ABB RobotStudio station: 实验二加基本自定义动作.rspag

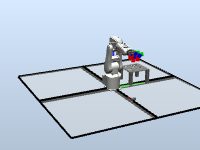
--- station ---
Station PartC (saved by RobotStudio 6.8.8148.134)
Controller System2
  mechanical unit ROB_1: IRB120_3_58__01, 6 joints, base frame (0, 0, 0) mm
Layout (positions relative to the parent item):
  - IRB120_3_58__01 [mechanism, from Robots\IRB120_3_58_G_01.rslib] at (0, 0, 0) mm; joint values [0.0061, 0.1198, 0.0289, 0.0001, -0.1484, -0.0004] (rad or m)
  - SmartComponent_1 [smart component] at (413.29, 2.5, 582.55) mm, rotated rx -130.44 ry 89.98 rz -130.09 deg
      signals: DI GET, DO FINISH, DI GET1, DO FINISH1
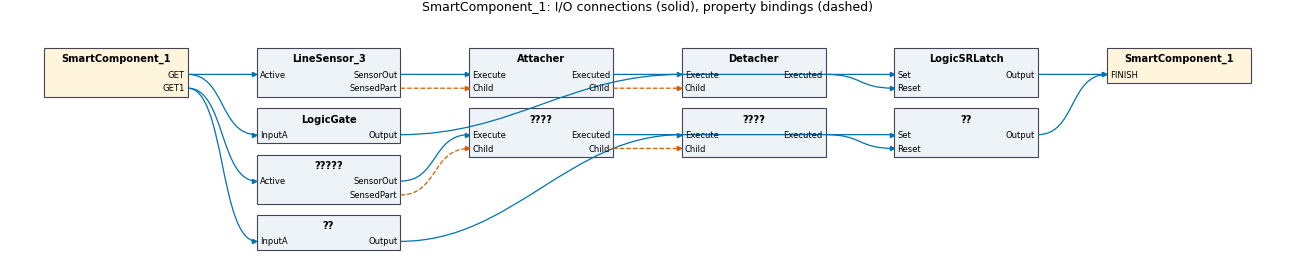
      connections:
        SmartComponent_1.GET -> LineSensor_3.Active
        SmartComponent_1.GET -> LogicGate.InputA
        LineSensor_3.SensorOut -> Attacher.Execute
        LogicGate.Output -> Detacher.Execute
        Attacher.Executed -> LogicSRLatch.Set
        Detacher.Executed -> LogicSRLatch.Reset
        LogicSRLatch.Output -> SmartComponent_1.FINISH
        SmartComponent_1.GET1 -> 吸盘传感器.Active
        SmartComponent_1.GET1 -> 吸盘.InputA
        吸盘传感器.SensorOut -> 吸盘安装.Execute
        吸盘.Output -> 吸盘拆除.Execute
        吸盘安装.Executed -> 吸盘.Set
        吸盘拆除.Executed -> 吸盘.Reset
        吸盘.Output -> SmartComponent_1.FINISH
        LineSensor_3.SensedPart => Attacher.Child
        Attacher.Child => Detacher.Child
        吸盘传感器.SensedPart => 吸盘安装.Child
        吸盘安装.Child => 吸盘拆除.Child
    - LineSensor_3 [smart component, from Components\LineSensor.rslib] at (-22.5, 0, 83.55) mm
        properties: Start=[0.0150000000000009 -0.000761999999999613 0.00306099999999904]; End=[-0.0249959999999991 0.00111800000000039 0.00431999999999905]; Radius=0.005; SensedPart=TCP-练习笔; SensedPoint=[-0.0910473251342774 0.454946044921875 0.202438980102539]
      - _sensorPart_ [part]
    - Attacher [smart component, from Components\Attacher.rslib]
        properties: Parent=SmartComponent_1; Flange=0; Child=TCP-练习笔; Mount=false; Offset=[0 0 0]; Orientation=[0 0 0]
    - Detacher [smart component, from Components\Detacher.rslib]
        properties: Child=TCP-练习笔; KeepPosition=true
    - LogicGate [smart component, from Components\LogicGate.rslib]
        properties: Operator=NOT; Delay=0
    - LogicSRLatch [smart component, from Components\LogicSRLatch.rslib]
    - My_Mechanism [mechanism] at (0, 0, 0) mm; joint values [0.01] (rad or m)
        TCP tool1 at (15.5, 0, 69.3) mm
        TCP tool2 at (-22.5, 0, 83.55) mm
        TCP tool3 at (-22.5, 0, 160.55) mm
        links: L1, L2
    - 吸盘传感器 [smart component, from Components\LineSensor.rslib] at (15.5, 0, 69.3) mm
        properties: Start=[-9.24038488097009E-05 3.65283253372798E-07 6.91615849535143E-07]; End=[0.00653224996369399 -0.000166814998235508 -0.000226620747395823]; Radius=0.005; SensedPart=部件_2; SensedPoint=[0.465495025634766 0.029700740814209 0.03]
      - _sensorPart_ [part]
    - 吸盘安装 [smart component, from Components\Attacher.rslib]
        properties: Parent=SmartComponent_1; Flange=0; Child=部件_2; Mount=false; Offset=[0 0 0]; Orientation=[0 0 0]
    - 吸盘拆除 [smart component, from Components\Detacher.rslib]
        properties: Child=部件_2; KeepPosition=true
    - 吸盘 [smart component, from Components\LogicGate.rslib]
        properties: Operator=NOT; Delay=0
    - 吸盘 [smart component, from Components\LogicSRLatch.rslib]
  - 部件_2 [part] at (0, 0, 0) mm
  - TCP_Table [part]
  - TCP-练习笔 [part] at (0, 0, 0) mm
  - 框架_1 [frame] at (15.5, 0, 69.3) mm
  - 框架_2 [frame] at (-22.5, 0, 83.55) mm
  - 框架_3 [frame] at (-22.5, 0, 160.55) mm
Attachment: My_Mechanism is attached to IRB120_3_58__01 / Link6
Attachment: SmartComponent_1 is attached to IRB120_3_58__01 / Link6
Attachment: LineSensor_3 is attached to My_Mechanism / L1
Attachment: 吸盘传感器 is attached to My_Mechanism / L1
EventTableEntry 2443: Group=, Trigger=DO_007 2444, Actions=[EventTableActionMechanicalPose 2445], Comment=, ActivationMode=2, Cyclic=false
EventTableTriggerIO 2444: IOValue=[1], IRC5Controller=? -1, Operator=0, SignalSource=System2 2451
EventTableActionMechanicalPose 2445: VirtualSignal=, Mechanism=My_Mechanism 980, ToPoseName=SyncPosition, VirtualSignalValue=[1]
EventTableEntry 2446: Group=, Trigger=DO_007 2447, Actions=[EventTableActionMechanicalPose 2448], Comment=, ActivationMode=2, Cyclic=false
EventTableTriggerIO 2447: IOValue=[0], IRC5Controller=? -1, Operator=0, SignalSource=System2 2451
EventTableActionMechanicalPose 2448: VirtualSignal=, Mechanism=My_Mechanism 980, ToPoseName=HomePosition, VirtualSignalValue=[1]
Station logic (signal -> signal, property => property):
  System2.DO_007 -> SmartComponent_1.GET
  System2.DO_0077 -> SmartComponent_1.GET1
Targets, tools, work objects and paths stored in the station and not in the controller backup, written as RAPID:
! task T_ROB1
MODULE CalibData
  PERS tooldata tool1:=[TRUE,[[15.5,0,69.3],[1,0,0,0]],[1,[0,0,1],[1,0,0,0],0,0,0]];
  PERS tooldata tool2:=[TRUE,[[-22.5,0,83.554],[1,0,0,0]],[1,[0,0,1],[1,0,0,0],0,0,0]];
  PERS tooldata tool3:=[TRUE,[[-22.5,0,160.554],[1,0,0,0]],[1,[0,0,1],[1,0,0,0],0,0,0]];
  PERS tooldata Tooldata_4:=[TRUE,[[15.5,0,69.3],[1,0,0,0]],[1,[0,0,1],[1,0,0,0],0,0,0]];
  PERS tooldata Tooldata_5:=[TRUE,[[-22.5,0,83.554],[1,0,0,0]],[1,[0,0,1],[1,0,0,0],0,0,0]];
  PERS tooldata Tooldata_6:=[TRUE,[[-22.5,0,160.554],[1,0,0,0]],[1,[0,0,1],[1,0,0,0],0,0,0]];
ENDMODULE


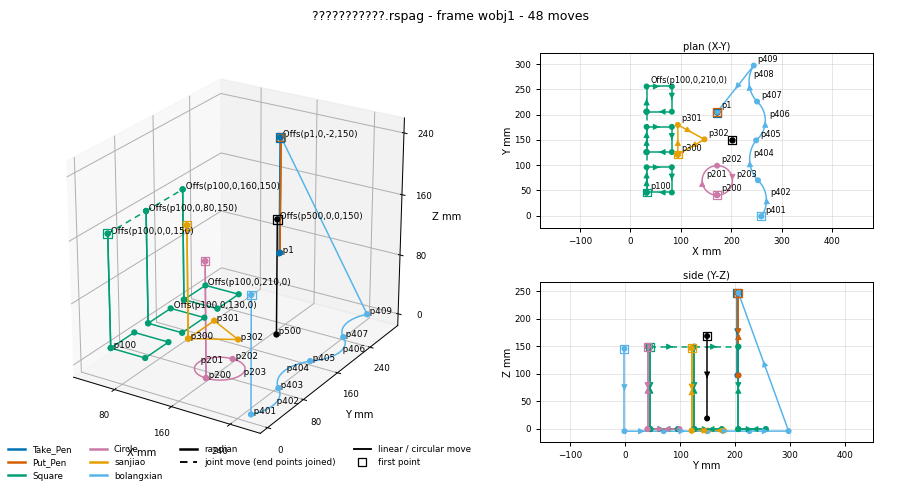
[picture p0: tool path of 实验二加基本自定义动作.rspag in frame wobj1, 48 of 55 moves have a stored position in this frame; points joined in program order, loops and branches not executed]
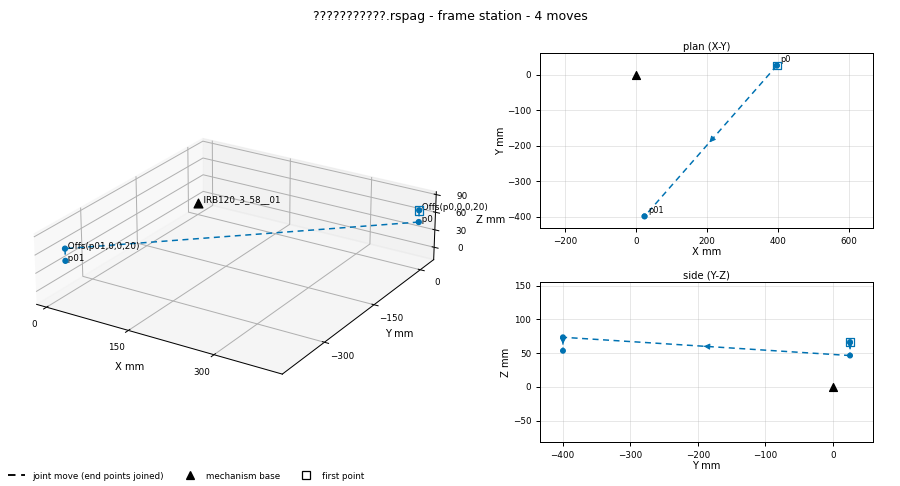
[picture p1: tool path of 实验二加基本自定义动作.rspag in frame station, 4 of 55 moves have a stored position in this frame; points joined in program order, loops and branches not executed]
--- Backups/System2/RAPID/TASK1/PROGMOD/Module1.mod ---
MODULE Module1
	TASK PERS loaddata load1:=[1,[0,0,50],[1,0,0,0],0,0,0];
	CONST robtarget p1:=[[172.01,205.77,97.31],[0.00112688,-0.706761,0.707451,0.00098463],[1,-1,0,0],[9E+9,9E+9,9E+9,9E+9,9E+9,9E+9]];
	CONST robtarget p100:=[[31.94,45.61,-0.49],[0.00223608,-0.000486235,-0.999989,-0.00403198],[1,-1,0,0],[9E+9,9E+9,9E+9,9E+9,9E+9,9E+9]];
	CONST robtarget p200:=[[171.47,40.35,-0.47],[0.00223616,-0.000486939,-0.999989,-0.00403224],[1,0,0,0],[9E+9,9E+9,9E+9,9E+9,9E+9,9E+9]];
	CONST robtarget p201:=[[142.00,69.14,-0.45],[0.00223618,-0.000487262,-0.999989,-0.00403234],[1,0,0,0],[9E+9,9E+9,9E+9,9E+9,9E+9,9E+9]];
	CONST robtarget p202:=[[171.58,98.63,-0.43],[0.00223622,-0.000487166,-0.999989,-0.0040324],[1,0,0,0],[9E+9,9E+9,9E+9,9E+9,9E+9,9E+9]];
	CONST robtarget p203:=[[201.97,69.09,-0.44],[0.00223617,-0.000487189,-0.999989,-0.00403229],[1,0,0,0],[9E+9,9E+9,9E+9,9E+9,9E+9,9E+9]];
	CONST robtarget p0:=[[396.39,25.44,46.35],[0.705985,-0.0237396,0.707527,0.0206965],[0,0,-1,1],[9E+9,9E+9,9E+9,9E+9,9E+9,9E+9]];
	CONST robtarget p01:=[[23.64,-399.51,53.40],[0.514651,0.477849,0.513743,-0.49281],[-1,0,-1,1],[9E+9,9E+9,9E+9,9E+9,9E+9,9E+9]];
	CONST robtarget p300:=[[93.84,120.75,-3.23],[0.00223478,-0.000452817,-0.999989,-0.0040181],[1,0,0,0],[9E+9,9E+9,9E+9,9E+9,9E+9,9E+9]];
	CONST robtarget p301:=[[93.89,179.47,-3.19],[0.0022349,-0.00045269,-0.999989,-0.00401838],[1,0,0,0],[9E+9,9E+9,9E+9,9E+9,9E+9,9E+9]];
	CONST robtarget p302:=[[146.61,150.84,-3.20],[0.00223477,-0.000452827,-0.999989,-0.00401803],[1,0,0,0],[9E+9,9E+9,9E+9,9E+9,9E+9,9E+9]];
	CONST robtarget p401:=[[259.28,-1.69,-4.25],[0.00223475,-0.000452484,-0.999989,-0.00401722],[1,0,0,0],[9E+9,9E+9,9E+9,9E+9,9E+9,9E+9]];
	CONST robtarget p402:=[[269.21,32.94,-4.22],[0.00223475,-0.000454397,-0.999989,-0.00401611],[0,0,-1,0],[9E+9,9E+9,9E+9,9E+9,9E+9,9E+9]];
	CONST robtarget p403:=[[252.60,69.70,-4.20],[0.00223474,-0.000455037,-0.999989,-0.00401594],[1,0,0,0],[9E+9,9E+9,9E+9,9E+9,9E+9,9E+9]];
	CONST robtarget p404:=[[236.03,109.91,-4.18],[0.00223473,-0.00045505,-0.999989,-0.00401592],[1,0,0,0],[9E+9,9E+9,9E+9,9E+9,9E+9,9E+9]];
	CONST robtarget p405:=[[248.98,148.90,-4.15],[0.00223474,-0.000454835,-0.999989,-0.00401611],[1,0,0,0],[9E+9,9E+9,9E+9,9E+9,9E+9,9E+9]];
	CONST robtarget p406:=[[267.17,187.83,-4.12],[0.00223473,-0.000455175,-0.999989,-0.00401622],[0,0,-1,0],[9E+9,9E+9,9E+9,9E+9,9E+9,9E+9]];
	CONST robtarget p407:=[[250.72,225.76,-4.10],[0.00223473,-0.000455584,-0.999989,-0.00401679],[1,0,0,0],[9E+9,9E+9,9E+9,9E+9,9E+9,9E+9]];
	CONST robtarget p408:=[[234.94,267.04,-4.07],[0.00223476,-0.000456023,-0.999989,-0.00401721],[1,0,0,0],[9E+9,9E+9,9E+9,9E+9,9E+9,9E+9]];
	CONST robtarget p409:=[[244.29,297.08,-4.05],[0.00223476,-0.000455568,-0.999989,-0.00401737],[1,0,0,0],[9E+9,9E+9,9E+9,9E+9,9E+9,9E+9]];
	CONST robtarget p500:=[[202.00,148.79,18.91],[0.00223468,-0.000457037,-0.999989,-0.00401663],[1,0,0,0],[9E+9,9E+9,9E+9,9E+9,9E+9,9E+9]];
	VAR num pCenter:=0;
    !***********************************************************
    !
    ! Module:  Module1
    !
    ! Description:
    !   <Insert description here>
    !
    ! Author: He
    !
    ! Version: 1.0
    !
    !***********************************************************


    !***********************************************************
    !
    ! Procedure main
    !
    !   This is the entry point of your program
    !
    !***********************************************************
    PROC main()
        Reset DO_007;
        Reset DO_0077;
        xipan;
        Initialize;
        Take_Pen;
        Square;
        sanjiao;
        Circle;
        bolangxian;
        Put_Pen;
    ENDPROC
	PROC Initialize()
		AccSet 100, 100;
		VelSet 100, 300;
		MoveAbsJ [[0,0,0,0,0,0],[9E+9,9E+9,9E+9,9E+9,9E+9,9E+9]]\NoEOffs, v300, z50, tool0;
		MoveAbsJ [[90,0,0,0,90,0],[9E+9,9E+9,9E+9,9E+9,9E+9,9E+9]]\NoEOffs, v100, z50, tool0;
	ENDPROC
	PROC Take_Pen()
		MoveJ Offs(p1,0,-2,150), v100, z50, tool0\WObj:=wobj1;
		MoveL Offs(p1,0,-2,0), v50, fine, tool0\WObj:=wobj1;
		MoveL p1, v50, fine, tool0\WObj:=wobj1;
		Set DO_007;
		WaitTime 1;
		MoveL Offs(p1,0,0,150), v100, z50, tool0\WObj:=wobj1;
	ENDPROC
	PROC Put_Pen()
		MoveJ Offs(p1,0,0,150), v100, z50, tool0\WObj:=wobj1;
		MoveL p1, v50, fine, tool0\WObj:=wobj1;
		Reset DO_007;
		WaitTime 1;
		MoveL Offs(p1,0,0,150), v100, z50, tool0\WObj:=wobj1;
	ENDPROC
	PROC Square()
		!1
        MoveJ Offs(p100,0,0,150), v100, z50, tool_pen\WObj:=wobj1;
		MoveL p100, v50, fine, tool_pen\WObj:=wobj1;
		MoveL Offs(p100,0,50,0), v100, z50, tool_pen\WObj:=wobj1;
		MoveL Offs(p100,50,50,0), v100, z50, tool_pen\WObj:=wobj1;
		MoveL Offs(p100,50,0,0), v100, z50, tool_pen\WObj:=wobj1;
		MoveL p100, v100, fine, tool_pen\WObj:=wobj1;
		MoveL Offs(p100,0,0,150), v100, z50, tool_pen\WObj:=wobj1;
        !2
        MoveJ Offs(p100,0,80,150), v100, z50, tool_pen\WObj:=wobj1;
		MoveL Offs(p100,0,80,0), v50, fine, tool_pen\WObj:=wobj1;
		MoveL Offs(p100,0,130,0), v100, z50, tool_pen\WObj:=wobj1;
		MoveL Offs(p100,50,130,0), v100, z50, tool_pen\WObj:=wobj1;
		MoveL Offs(p100,50,80,0), v100, z50, tool_pen\WObj:=wobj1;
		MoveL Offs(p100,0,80,0), v100, fine, tool_pen\WObj:=wobj1;
		MoveL Offs(p100,0,80,150), v100, z50, tool_pen\WObj:=wobj1;
        !3
        MoveJ Offs(p100,0,160,150), v100, z50, tool_pen\WObj:=wobj1;
		MoveL Offs(p100,0,160,0), v50, fine, tool_pen\WObj:=wobj1;
		MoveL Offs(p100,0,210,0), v100, z50, tool_pen\WObj:=wobj1;
		MoveL Offs(p100,50,210,0), v100, z50, tool_pen\WObj:=wobj1;
		MoveL Offs(p100,50,160,0), v100, z50, tool_pen\WObj:=wobj1;
		MoveL Offs(p100,0,160,0), v100, fine, tool_pen\WObj:=wobj1;
		MoveL Offs(p100,0,160,150), v100, z50, tool_pen\WObj:=wobj1;
	ENDPROC
	PROC Circle()
		MoveJ Offs(p200,0,0,150), v100, z50, tool_pen\WObj:=wobj1;
		MoveL p200, v50, fine, tool_pen\WObj:=wobj1;
		MoveC p201, p202, v100, z50, tool_pen\WObj:=wobj1;
		MoveC p203, p200, v100, fine, tool_pen\WObj:=wobj1;
		MoveL Offs(p200,0,0,150), v100, z10, tool_pen\WObj:=wobj1;
	ENDPROC
	PROC xipan()
		MoveAbsJ [[0,0,0,0,0,0],[9E+9,9E+9,9E+9,9E+9,9E+9,9E+9]]\NoEOffs, v100, z50, tool0;
		MoveJ Offs(p0,0,0,20), v100, fine, tool0\WObj:=wobj0;
		MoveJ p0, v100, fine, tool0;
		WaitTime 1;
		Set DO_0077;
		WaitTime 1;
		MoveJ Offs(p01,0,0,20), v100, fine, tool0;
		MoveJ p01, v100, fine, tool0;
		Reset DO_0077;
		WaitTime 1;
	ENDPROC
	PROC sanjiao()
		MoveJ Offs(p300,0,0,150), v100, z50, tool_pen\WObj:=wobj1;
		MoveL p300, v50, fine, tool_pen\WObj:=wobj1;
		MoveL p301, v100, z50, tool_pen\WObj:=wobj1;
		MoveL p302, v100, z50, tool_pen\WObj:=wobj1;
		MoveL p300, v100, fine, tool_pen\WObj:=wobj1;
		MoveL Offs(p300,0,0,150), v100, z50, tool_pen\WObj:=wobj1;
	ENDPROC
	PROC bolangxian()
		MoveJ Offs(p401,0,0,150), v100, z50, tool_pen\WObj:=wobj1;
		MoveL p401, v50, fine, tool_pen\WObj:=wobj1;
		MoveC p402, p403, v100, z50, tool_pen\WObj:=wobj1;
		MoveC p404, p405, v100, fine, tool_pen\WObj:=wobj1;
        MoveC p406, p407, v100, z50, tool_pen\WObj:=wobj1;
		MoveC p408, p409, v100, fine, tool_pen\WObj:=wobj1;
		MoveL Offs(p1,0,0,150), v100, z10, tool0\WObj:=wobj1;
	ENDPROC
	PROC raodian()
		MoveJ Offs(p500,0,0,150), v100, z50, tool_pen\WObj:=wobj1;
        MoveL p500, v100, fine, tool_pen\WObj:=wobj1;
        FOR i FROM 0 TO 360 STEP 10 DO
        	pCenter := <EXP>;
        ENDFOR
	ENDPROC
ENDMODULE

--- Backups/System2/SYSPAR/EIO.cfg ---
EIO:CFG_1.0:6:1::
#
INDUSTRIAL_NETWORK:

      -Name "DeviceNet" -Label "DeviceNet Master/Slave Network" -Address "2"
#
DEVICENET_DEVICE:

      -Name "d652" -VendorName "ABB Robotics" -ProductName "24 VDC I/O Device"\
      -Label "DSQC 652 24 VDC I/O Device" -Address 10 -ProductCode 26\
      -DeviceType 7 -ConnectionType "COS" -OutputSize 2 -InputSize 2
#
DEVICENET_INTERNAL_DEVICE:

      -Name "DN_Internal_Device" -VendorName "ABB Robotics"\
      -ProductName "DeviceNet Internal Slave Device"
#
EIO_SIGNAL:

      -Name "DO_007" -SignalType "DO" -Device "d652" -DeviceMap "7"

      -Name "DO_0077" -SignalType "DO" -Device "d652" -DeviceMap "1"
